FUNCTION_BLOCK FB_Linked_List
VAR_INPUT
END_VAR
VAR_OUTPUT
END_VAR
VAR
	pHead :  POINTER TO ST_NODE;
	pTail :  POINTER TO ST_NODE;
END_VAR

// Adds an node to the end of the linked list
METHOD Create
VAR_INPUT
	Data : T_DATA_TYPE;
END_VAR
VAR
	pTemp :  POINTER TO ST_NODE;
END_VAR
pTemp := __NEW(ST_NODE); 	// Allocate space in memory for a node.
pTemp^.Data := Data;		// Assign Data to the new node.
pTemp^.pNext := NULL;		// Pointer to next node is NULL.
IF pHead = 0 THEN pHead := pTemp; pTail := pTemp; // If the pointer to the pHead is NULL then give it an address. The pTail address of the first node is the pHead.
ELSE  pTail^.pNext := pTemp; pTail := pTail^.pNext; END_IF // Point previous node's pNext to the address of pTemp and set pTail to pTemp.
END_METHOD

// Traverse the list to display each node
METHOD Display
VAR_IN_OUT
	aList 		: ARRAY[*] OF T_DATA_TYPE;
END_VAR
VAR
	pCurrent 	:  POINTER TO ST_NODE;
	i 			: DINT;
END_VAR
pCurrent := pHead;
i := LOWER_BOUND(aList, 1);
WHILE pCurrent <> 0 AND i < UPPER_BOUND(aList, 1) DO
	aList[i] := pCurrent^.Data;
	pCurrent := pCurrent^.pNext;
	i := i+1;
END_WHILE
END_METHOD

// Initializes or create an empty list
METHOD Init
pHead := NULL;
pTail := NULL;
END_METHOD

// Inserts node at a specific position in the list
METHOD Insert
VAR_INPUT
	Data 		: T_DATA_TYPE;
	nPosition 	: UXINT; 
END_VAR
VAR
	pPrevious 	: POINTER TO ST_NODE;
	pCurrent 	: POINTER TO ST_NODE;
	pTemp 		: POINTER TO ST_NODE;
	i 			: UXINT;
END_VAR
// Create new node
//pPrevious := __NEW(ST_NODE);
//pCurrent := __NEW(ST_NODE); 	
pTemp := __NEW(ST_NODE);

pCurrent := pHead;
FOR i := 1 TO nPosition DO
	pPrevious := pCurrent;
	pCurrent := pPrevious^.pNext;
	END_FOR;
pTemp^.Data := Data;
pPrevious^.pNext := pTemp;
pTemp^.pNext := pCurrent;
END_METHOD

// Deletes/pops a node at the start of the list 
METHOD Pop
VAR
	pTemp : POINTER TO ST_NODE;
END_VAR
pTemp := pHead^.pNext;
__DELETE(pHead);
pHead := pTemp;
END_METHOD

// Adds/pushes a node at the start of the list 
METHOD Push
VAR_INPUT
	Data 	: T_DATA_TYPE;
END_VAR
VAR
	pTemp 	:  POINTER TO ST_NODE;
END_VAR
pTemp := __NEW(ST_NODE); 	// Allocate space in memory for a node.
pTemp^.Data := Data;
pTemp^.pNext := pHead;
pHead := pTemp;
END_METHOD

END_FUNCTION_BLOCK

(* stored: Version 1.1.0.1, ProductVersion 3.1.4024.4
   POU FB_Linked_List: Id {19223dee-072c-4cbb-9e58-eedc7741ea7e}, SpecialFunc None
   Method Create: Id {1c02436b-f1d7-46b9-bde8-e418c191c48f}
   Method Display: Id {44cc05c3-a73a-485e-b7c4-9f46d1a3c88e}
   Method Init: Id {d3845c5b-4488-4a2a-83ef-21fe8d01c1da}
   Method Insert: Id {b50ffa90-bffd-42d6-880d-1e20342d73fd}
   Method Pop: Id {a3623de3-4c8b-4ca0-a7a5-e2d659fad6d5}
   Method Push: Id {fc4a9c4f-82e1-46e6-8281-109c5a2f41f3} *)
